// TIA Portal V16 export
// export: Created 2022-02-04T14:40:20.3341903Z, ExportSetting WithDefaults, DisplayName Totally Integrated Automation Portal, DisplayVersion V16 Update 1, DisplayName TIA Portal Version Control Interface, DisplayVersion V16, DisplayName TIA Portal Openness, DisplayVersion V16, DisplayName SINAMICS Startdrive Advanced, DisplayVersion V16 Update 5, DisplayName SINAMICS Startdrive G130, G150, S120, S150, SINAMICS MV, S210, DisplayVersion V16 Update 5, DisplayName SINAMICS Startdrive G110M, G120, G120C, G120D, G120P, G115D, DisplayVersion V16 Update 5, DisplayName STEP 7 Professional, DisplayVersion V16, DisplayName STEP 7 Safety, DisplayVersion V16, DisplayName WinCC Advanced, DisplayVersion V16, DisplayName SIMATIC Visualization Architect, DisplayVersion V16
DATA_BLOCK "MovableBoard_CTRL_DB"   // DB13
VERSION : 0.1
// stored: AutoNumber true, InstanceOfName MovableBoard_CTRL, InstanceOfType FB
"MovableBoard_CTRL"
   // VAR_INPUT
   //    BoardBase : Bool;
   //    ModeChanged : Bool;
   //    Reset : Bool;
   //    EncPos : Byte;
   //    SetPos : Int;
   // END_VAR
   // VAR_OUTPUT
   //    CMD_Fwd : Bool;
   //    CMD_Bwd : Bool;
   //    CMD_UP : Bool;
   //    CMD_DOWN : Bool;
   //    AutoMode : Bool;
   //    ResetVirtualPos : Bool;
   //    Position : Int;
   // END_VAR
   // VAR RETAIN
   //    DefinitionTag : Bool;
   //    ChangingPos : Bool;
   //    ShutUpAuto : Bool;
   //    startOffset : Int;
   //    curMicroPos : Int;
   //    curMicroPos_old : Int;
   //    curMacroPos : Int;
   // END_VAR
BEGIN
END_DATA_BLOCK
